Fanuc KAREL source: kd00073.KL

-- PROVISIONAL review KL for V940-1; original PC SHA256 415abfc21f2c46cd1cad32f0c35d209152f9ebe2cefdba860575eb7bcf738a63
-- Incomplete behavior may be omitted. Consult companion uncertainty JSON. Do not deploy.
PROGRAM KD00073
%NOLOCKGROUP
VAR
  I : INTEGER
  J : INTEGER
  B : BOOLEAN
  R : REAL
  S : STRING[80]
BEGIN
  -- V9_EXPOSED_INDEXED_TABLE_HINT layout=0001; 1 counted words exposed once; source arms/runtime held
  -- UNRESOLVED_PC offsets 5-12; opcodes 9C,23
  -- UNRESOLVED_PC offsets 22-36; opcodes 21,9D,52,23
  -- UNRESOLVED_PC offsets 41-58; opcodes 21,2E,5B,79
  -- UNRESOLVED_PC offsets 63-67; opcodes 7F
END KD00073
